INTERFACE ILog

METHOD SetLogger : BOOL
VAR_INPUT
    ref2Core : LogCore;
END_VAR
END_METHOD

END_INTERFACE

(* stored: Version 1.1.0.1
   Itf ILog: Id {142e5ac4-9651-4b60-842f-9fed1e0c8704}
   Method SetLogger: Id {3e80fdb5-b4db-45a7-930c-3a38b44c5bfc} *)
